PROGRAM MAIN
VAR
	
bool1				:	BOOL;

deskbool			:	BOOL;

lapbool				:	BOOL;

mainBranchLapBool2	:	BOOL;

mainBranchLapBool3	:	BOOL;

END_VAR

END_PROGRAM

(* stored: Version 1.1.0.1, ProductVersion 3.1.4024.12
   POU MAIN: Id {82f0ea0d-1406-4204-9446-c1968db403d4}, SpecialFunc None *)
